FUNCTION_BLOCK PLCnextAXLSEDO16 (* Service Interface Function Block Type *)
  (* Standard: 61499-2; Description: Copyright (c) 2022 Peirlberger Juergen This program and the accompanying materials are made available under the terms of the Eclipse Public License 2.0 which is available at https://www.eclipse.org/legal/epl-2.0/ SPDX-License-Identifier: EPL-2.0 *)
  (* Version 1.0, 2022-04-07, Peirlberger Juergen *)
  (* Version 3.0, 2025-04-14, Patrick Aigner, changed package *)
  PACKAGE eclipse4diac::io::plcnext;
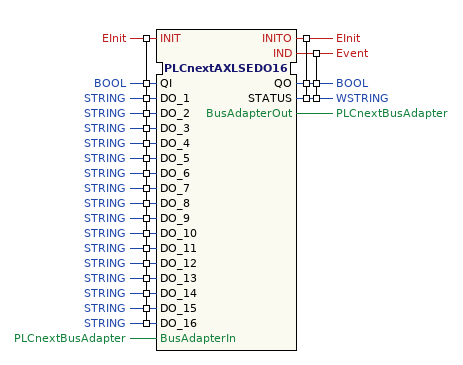
  EVENT_INPUT
    INIT : EInit WITH QI, DO_1, DO_2, DO_3, DO_4, DO_5, DO_6, DO_7, DO_8, DO_9, DO_10, DO_11, DO_12, DO_13, DO_14, DO_15, DO_16; (* Service Initialization *)
  END_EVENT
  EVENT_OUTPUT
    INITO : EInit WITH QO, STATUS; (* Initialization Confirm *)
    IND WITH QO, STATUS; (* Indication from Resource *)
  END_EVENT
  VAR_INPUT
    QI : BOOL; (* Event Input Qualifier *)
    DO_1 : STRING := ''; (* Digital Output *)
    DO_2 : STRING; (* Digital Output *)
    DO_3 : STRING; (* Digital Output *)
    DO_4 : STRING; (* Digital Output *)
    DO_5 : STRING; (* Digital Output *)
    DO_6 : STRING; (* Digital Output *)
    DO_7 : STRING; (* Digital Output *)
    DO_8 : STRING; (* Digital Output *)
    DO_9 : STRING; (* Digital Output *)
    DO_10 : STRING; (* Digital Output *)
    DO_11 : STRING; (* Digital Output *)
    DO_12 : STRING; (* Digital Output *)
    DO_13 : STRING; (* Digital Output *)
    DO_14 : STRING; (* Digital Output *)
    DO_15 : STRING; (* Digital Output *)
    DO_16 : STRING; (* Digital Output *)
  END_VAR
  VAR_OUTPUT
    QO : BOOL; (* Event Output Qualifier *)
    STATUS : WSTRING; (* Service Status *)
  END_VAR
  SOCKETS
    BusAdapterIn : eclipse4diac::io::plcnext::PLCnextBusAdapter;
  END_SOCKETS
  PLUGS
    BusAdapterOut : eclipse4diac::io::plcnext::PLCnextBusAdapter;
  END_PLUGS
END_FUNCTION_BLOCK
